PROGRAM MAIN
VAR
	bON: BOOL; 
	bOFF: BOOL;
END_VAR

(*
  	  ESCOLA POLITÉCNICA DE ENXEÑARÍA DE FERROL			
			  UNIVERSIDADE DA CORUÑA 						
			
Máster Universitario en Informática Industrial y Robótica   
  	Automatización Avanzada - Curso 2023-2024			

					Profesorado: 						
 	Antonio J. Díaz Longueira - Míriam Timiraos Díaz 		

 		    	Código realizado por:
	Marta María Álvarez Crespo - Noelia Pita López  		
*)

PRG_LlenadoCajas();
POU_StopBladePyP();
POU_Contadores();
PRG_Turntable();
PRG_Almacen();

IF GVL_General.bMarcha THEN
	bON := TRUE;
END_IF

IF GVL_General.bParo THEN
	bOFF := TRUE;
END_IF

IF bON AND NOT bOFF AND GVL_General.bSetaEmergencia THEN
	POU_OnFabrica();
	POU_ProcesoEntrada();
	POU_PickAndPlace();
	POU_PositionerAzul();
	POU_Parada();
END_IF

IF bOFF THEN
	POU_FinDeCiclo();
	bON := FALSE;
END_IF

IF NOT GVL_General.bSetaEmergencia THEN
	POU_SetaEmergencia();
END_IF































































(*
		♡ 
    /\_____/\
   /  o   o  \						
  ( ==  ^  == )		
   )         (		   __     miau
 (             )______/  |		miau 
(__(__)___(__)__)_______/	 

*)

END_PROGRAM

(* stored: Version 1.1.0.1, ProductVersion 3.1.4024.12
   POU MAIN: Id {28e20df2-0591-4dfb-a4d7-597d7dcfe426}, SpecialFunc None *)
